FUNCTION Convert_DINT_TO_DT : Hresult
VAR_INPUT
	in : DINT;
	out : REFERENCE TO DT;
END_VAR
VAR
	converted : DT;
END_VAR
VAR CONSTANT
	INCOMPATIBLE : HRESULT := 16#9811070E;
END_VAR

converted := DINT_TO_DT(in);

IF (DT_TO_DINT(converted) <> in) THEN
	Convert_DINT_TO_DT := INCOMPATIBLE;
	RETURN;
END_IF

out := converted;

END_FUNCTION

(* stored: Version 1.1.0.1, ProductVersion 3.1.4024.12
   POU Convert_DINT_TO_DT: Id {75297413-c549-4883-b873-87a1b1abcb86}, SpecialFunc None *)
